// TIA Portal V17 export
// export: Created 2025-06-26T06:49:24.6875755Z, ExportSetting WithDefaults, DisplayName Totally Integrated Automation Portal, DisplayVersion V17 Update 8, DisplayName TIA Portal Openness, DisplayVersion V17 Update 8, DisplayName TIA Portal Version Control Interface, DisplayVersion V17, DisplayName STEP 7 Professional, DisplayVersion V17 Update 8, DisplayName STEP 7 Safety, DisplayVersion V17 Update 6, DisplayName WinCC Advanced, DisplayVersion V17 Update 8
DATA_BLOCK "DB_Alarms"   // DB44
{ S7_Optimized_Access := 'FALSE' }
AUTHOR : Heaten
VERSION : 0.1
// stored: AutoNumber true, DBAccessibleFromOPCUA true, DBAccessibleFromWebserver true, IsOnlyStoredInLoadMemory false, IsWriteProtectedInAS false
   VAR RETAIN
      bAckAll : Bool := FALSE;   // Global alarm acknowledge
      bCommonAlarm : Bool := FALSE;   // Global common alarm
      bCriticalAlarm : Bool := FALSE;   // Global critical alarm
      "0001_WatchdogTimeoutOB1" { S7_SetPoint := 'True'} : "stEvent";
      "0003_InitCurrentSettingsFailed" { S7_SetPoint := 'True'} : "stEvent";
      "1001_ConnectionToWinCClost" { S7_SetPoint := 'True'} : "stEvent";
      "1002_EmergencyStopActive" { S7_SetPoint := 'True'} : "stEvent";
      "1003_EmergencyStopResetFailed" { S7_SetPoint := 'True'} : "stEvent";
      "1004_HBL_PS_500_X2" { S7_SetPoint := 'True'} : "stEvent";
      "1101_HBL_SC_01_CommError" { S7_SetPoint := 'True'} : "stDigitalAlarm";
      "1102_HBL_SC_02_CommError" { S7_SetPoint := 'True'} : "stDigitalAlarm";
      "1103_HBL_SC_03_CommError" { S7_SetPoint := 'True'} : "stDigitalAlarm";
      "1110_HBL_SC_10_CommError" { S7_SetPoint := 'True'} : "stDigitalAlarm";
      "1121_HBL_SC_01_Tripped" { S7_SetPoint := 'True'} : "stDigitalAlarm";
      "1122_HBL_SC_02_Tripped" { S7_SetPoint := 'True'} : "stDigitalAlarm";
      "1123_HBL_SC_03_Tripped" { S7_SetPoint := 'True'} : "stDigitalAlarm";
      "1130_HBL_SC_10_Tripped" { S7_SetPoint := 'True'} : "stDigitalAlarm";
      "1140_HBL_SC_01_RunFailure" { S7_SetPoint := 'True'} : "stDigitalAlarm";
      "1142_HBL_SC_02_RunFailure" { S7_SetPoint := 'True'} : "stDigitalAlarm";
      "1143_HBL_SC_03_RunFailure" { S7_SetPoint := 'True'} : "stDigitalAlarm";
      "1150_HBL_SC_10_RunFailure" { S7_SetPoint := 'True'} : "stDigitalAlarm";
      "1201_HBL_PT_517_Fault" { S7_SetPoint := 'True'} : "stEvent";
      "1202_HBL_PT_612_Fault" { S7_SetPoint := 'True'} : "stEvent";
      "1203_HBL_PT_519_Fault" { S7_SetPoint := 'True'} : "stEvent";
      "1204_HBL_PT_544_Fault" { S7_SetPoint := 'True'} : "stEvent";
      "1205_HBL_TT_516_Fault" { S7_SetPoint := 'True'} : "stEvent";
      "1206_HBL_TT_611_Fault" { S7_SetPoint := 'True'} : "stEvent";
      "1207_HBL_TT_901_Fault" { S7_SetPoint := 'True'} : "stEvent";
      "1208_HBL_TT_518_Fault" { S7_SetPoint := 'True'} : "stEvent";
      "1209_HBL_HCV_576_A1_Fault" { S7_SetPoint := 'True'} : "stEvent";
      "1210_HBL_TT_573_Fault" { S7_SetPoint := 'True'} : "stEvent";
      "1212_HBL_TT_543_Fault" { S7_SetPoint := 'True'} : "stEvent";
      "1213_HBL_TT_546_Fault" { S7_SetPoint := 'True'} : "stEvent";
      "1214_HBL_TT_542_Fault" { S7_SetPoint := 'True'} : "stEvent";
      "1215_HBL_TT_571_Fault" { S7_SetPoint := 'True'} : "stEvent";
      "1216_HBL_TT_16_Fault" { S7_SetPoint := 'True'} : "stEvent";
      "1217_HBL_TT_17_Fault" { S7_SetPoint := 'True'} : "stEvent";
      "1218_HBL_TT_18_Fault" { S7_SetPoint := 'True'} : "stEvent";
      "1220_HBL_PT_960_Fault" { S7_SetPoint := 'True'} : "stEvent";
      "1221_HBL_PT_05_Fault" { S7_SetPoint := 'True'} : "stEvent";
      "1223_HBL_TT_03_Fault" { S7_SetPoint := 'True'} : "stEvent";
      "1224_HBL_TT_23_Fault" { S7_SetPoint := 'True'} : "stEvent";
      "1225_HBL_TT_24_Fault" { S7_SetPoint := 'True'} : "stEvent";
      "1226_HBL_TT_25_Fault" { S7_SetPoint := 'True'} : "stEvent";
      "1227_HBL_LT_610_Fault" { S7_SetPoint := 'True'} : "stEvent";
      "1228_HBL_TT_21_Fault" { S7_SetPoint := 'True'} : "stEvent";
      "1229_HBL_TT_22_Fault" { S7_SetPoint := 'True'} : "stEvent";
      "1230_HBL_LT_02_Fault" { S7_SetPoint := 'True'} : "stEvent";   // Deprecated
      "1231_HBL_HCV_578_A1_Fault" { S7_SetPoint := 'True'} : "stEvent";
      "1232_HBL_PT_503_Fault" { S7_SetPoint := 'True'} : "stEvent";
      "1233_HBL_TT_20_Fault" { S7_SetPoint := 'True'} : "stDigitalAlarm";
      "1234_HBL_PT_14_Fault" { S7_SetPoint := 'True'} : "stEvent";   // Deprecated
      "1235_HBL_PT_18_Fault" { S7_SetPoint := 'True'} : "stEvent";   // Deprecated
      "1236_HBL_PT_19_Fault" { S7_SetPoint := 'True'} : "stEvent";   // Deprecated
      "1237_HBL_PT_25_Fault" { S7_SetPoint := 'True'} : "stEvent";   // Deprecated
      "1238_HBL_TT_31_Fault" { S7_SetPoint := 'True'} : "stEvent";   // Deprecated
      "1239_HBL_TT_33_Fault" { S7_SetPoint := 'True'} : "stEvent";   // Deprecated
      "1240_HBL_TT_35_Fault" { S7_SetPoint := 'True'} : "stEvent";   // Deprecated
      "1241_HBL_HCV_576_Fault" { S7_SetPoint := 'True'} : "stEvent";
      "1242_HBL_HCV_578_Fault" { S7_SetPoint := 'True'} : "stEvent";
      "1243_HBL_PT_902_Fault" { S7_SetPoint := 'True'} : "stEvent";
      "1244_HBL_PT_572_Fault" { S7_SetPoint := 'True'} : "stEvent";
      "1245_HBL_PT_09_Fault" { S7_SetPoint := 'True'} : "stEvent";   // Deprecated
      "1246_HBL_PT_547_Fault" { S7_SetPoint := 'True'} : "stEvent";
      "1247_HBL_PT_541_Fault" { S7_SetPoint := 'True'} : "stEvent";
      "1248_HBL_PT_531_Fault" { S7_SetPoint := 'True'} : "stEvent";
      "1249_HBL_PT_701_Fault" { S7_SetPoint := 'True'} : "stEvent";
      "1251_HBL_PT_534_Fault" { S7_SetPoint := 'True'} : "stEvent";
      "1252_HBL_TT_540_Fault" { S7_SetPoint := 'True'} : "stEvent";
      "1253_HBL_TT_530_Fault" { S7_SetPoint := 'True'} : "stEvent";
      "1254_HBL_TT_533_Fault" { S7_SetPoint := 'True'} : "stEvent";
      "1255_HBL_CT_01_Fault" { S7_SetPoint := 'True'} : "stEvent";
      "1256_HBL_CT_615_Fault" { S7_SetPoint := 'True'} : "stEvent";
      "1257_HBL_CT_03_Fault" { S7_SetPoint := 'True'} : "stEvent";
      "1258_HBL_TT_26_Fault" { S7_SetPoint := 'True'} : "stEvent";
      "1259_HBL_TT_27_Fault" { S7_SetPoint := 'True'} : "stEvent";
      "1260_HBL_FT_520_Fault" { S7_SetPoint := 'True'} : "stEvent";
      "1262_HBL_TT_504_Fault" { S7_SetPoint := 'True'} : "stEvent";
      "1263_HBL_TT_34_Fault" { S7_SetPoint := 'True'} : "stEvent";
      "1264_HBL_PT_961_Fault" { S7_SetPoint := 'True'} : "stEvent";
      "1265_HBL_TT_502_Fault" { S7_SetPoint := 'True'} : "stEvent";
      "1266_HBL_LT_510_Fault" { S7_SetPoint := 'True'} : "stEvent";
      "1267_HBL_PT_511_Fault" { S7_SetPoint := 'True'} : "stEvent";
      "1268_HBL_TT_512_Fault" { S7_SetPoint := 'True'} : "stEvent";
      "1269_HBL_TT_532_Fault" { S7_SetPoint := 'True'} : "stEvent";
      "1270_HBL_AT_535_Fault" { S7_SetPoint := 'True'} : "stEvent";
      "1271_HBL_AT_545_Fault" { S7_SetPoint := 'True'} : "stEvent";
      "1272_HBL_PT_635_Fault" { S7_SetPoint := 'True'} : "stEvent";
      "1273_HBL_PT_636_Fault" { S7_SetPoint := 'True'} : "stEvent";
      "1274_HBL_LT_650_Fault" { S7_SetPoint := 'True'} : "stEvent";
      "1275_HBL_PT_651_Fault" { S7_SetPoint := 'True'} : "stEvent";
      "1276_HBL_PT_702_Fault" { S7_SetPoint := 'True'} : "stEvent";
      "1277_HBL_HCV_514_Fault" { S7_SetPoint := 'True'} : "stEvent";
      "1278_HBL_HCV_514_A1_Fault" { S7_SetPoint := 'True'} : "stEvent";
      "1279_HBL_HCV_515_Fault" { S7_SetPoint := 'True'} : "stEvent";
      "1280_HBL_HCV_515_A1_Fault" { S7_SetPoint := 'True'} : "stEvent";
      "1281_HBL_HCV_548_Fault" { S7_SetPoint := 'True'} : "stEvent";
      "1282_HBL_HCV_548_A1_Fault" { S7_SetPoint := 'True'} : "stEvent";
      "1283_HBL_HCV_575_Fault" { S7_SetPoint := 'True'} : "stEvent";
      "1284_HBL_HCV_575_A1_Fault" { S7_SetPoint := 'True'} : "stEvent";
      "1285_HBL_HCV_577_Fault" { S7_SetPoint := 'True'} : "stEvent";
      "1286_HBL_HCV_577_A1_Fault" { S7_SetPoint := 'True'} : "stEvent";
      "1287_HBL_HCV_579_Fault" { S7_SetPoint := 'True'} : "stEvent";
      "1288_HBL_HCV_579_A1_Fault" { S7_SetPoint := 'True'} : "stEvent";
      "1289_HBL_HCV_616_Fault" { S7_SetPoint := 'True'} : "stEvent";
      "1290_HBL_HCV_616_A1_Fault" { S7_SetPoint := 'True'} : "stEvent";
      "1291_HBL_HCV_700_Fault" { S7_SetPoint := 'True'} : "stEvent";
      "1292_HBL_HCV_700_A1_Fault" { S7_SetPoint := 'True'} : "stEvent";
      "1293_HBL_PT_618_Fault" { S7_SetPoint := 'True'} : "stEvent";
      "1294_HBL_LS_632_Fault" { S7_SetPoint := 'True'} : "stDigitalAlarm";
      "1295_HBL_LS_633_Fault" { S7_SetPoint := 'True'} : "stDigitalAlarm";
      "2018_HBL_PT_05_High" { S7_SetPoint := 'True'} : "stLimitAlarm";
      "2028_HBL_PT_17_Low" { S7_SetPoint := 'True'} : "stLimitAlarm";
      "2058_HBL_TT_03_Low" { S7_SetPoint := 'True'} : "stLimitAlarm";
      "2100_HBL_TT_03_High" { S7_SetPoint := 'True'} : "stLimitAlarm";
      "2101_HBL_TT_901_High" { S7_SetPoint := 'True'} : "stLimitAlarm";
      "2102_HBL_PT_503_High" { S7_SetPoint := 'True'} : "stLimitAlarm";
      "2103_HBL_TT_518_High" { S7_SetPoint := 'True'} : "stLimitAlarm";
      "2105_HBL_TT_546_High" { S7_SetPoint := 'True'} : "stLimitAlarm";
      "2106_HBL_TT_17_High" { S7_SetPoint := 'True'} : "stLimitAlarm";
      "2107_HBL_TT_16_High" { S7_SetPoint := 'True'} : "stLimitAlarm";
      "2108_HBL_TT_18_High" { S7_SetPoint := 'True'} : "stLimitAlarm";
      "2109_HBL_TT_20_High" { S7_SetPoint := 'True'} : "stLimitAlarm";
      "2110_HBL_TT_21_High" { S7_SetPoint := 'True'} : "stLimitAlarm";
      "2111_HBL_TT_22_High" { S7_SetPoint := 'True'} : "stLimitAlarm";
      "2112_HBL_LT_02_High" { S7_SetPoint := 'True'} : "stLimitAlarm";   // Deprecated
      "2113_HBL_CT_01_High" { S7_SetPoint := 'True'} : "stLimitAlarm";
      "2114_HBL_CT_615_High" { S7_SetPoint := 'True'} : "stLimitAlarm";
      "2115_HBL_PT_17_LowLow" { S7_SetPoint := 'True'} : "stLimitAlarm";
      "2116_HBL_PT_503_HighHigh" { S7_SetPoint := 'True'} : "stLimitAlarm";
      "2117_HBL_TT_542_Low" { S7_SetPoint := 'True'} : "stLimitAlarm";
      "2301_HeatSourceTempDropCritical" { S7_SetPoint := 'True'} : "stLimitAlarm";
      "2302_HeatSourceTempRiseCritical" { S7_SetPoint := 'True'} : "stLimitAlarm";
      "2303_SuperheatCompressor_High" { S7_SetPoint := 'True'} : "stLimitAlarm";
      "2304_SuperheatCompressor_Low" { S7_SetPoint := 'True'} : "stLimitAlarm";
      "2305_OilFilterDeltaP_High" { S7_SetPoint := 'True'} : "stLimitAlarm";
      "2306_OilFilterDeltaP_HighHigh" { S7_SetPoint := 'True'} : "stLimitAlarm";
      "2307_EvaporatorDischargePressureMeanValue" { S7_SetPoint := 'True'} : "stEvent";
      "2308_EvaporatorDischargePressureHigh" { S7_SetPoint := 'True'} : "stLimitAlarm";
      "2309_OilSeparatorStage1High" { S7_SetPoint := 'True'} : "stDigitalAlarm";
      "3020_SuperheatControlRegulatorFault" { S7_SetPoint := 'True'} : "stEvent";
      "3030_PinchControlRegulatorfault" { S7_SetPoint := 'True'} : "stEvent";
      "3400_HydrolockProtectionActive" { S7_SetPoint := 'True'} : "stEvent";
      "3401_DripPanLevelHigh" { S7_SetPoint := 'True'} : "stDigitalAlarm";
      "5000_OilHeatingActivationFailure" { S7_SetPoint := 'True'} : "stDigitalAlarm";
      "5001_OilHeatingDeactivationFailure" { S7_SetPoint := 'True'} : "stDigitalAlarm";
      "5200_CPC_LT_870_Fault" { S7_SetPoint := 'True'} : "stEvent";
      "5201_CPC_TT_871_Fault" { S7_SetPoint := 'True'} : "stEvent";
      "5202_CPC_PT_872_Fault" { S7_SetPoint := 'True'} : "stEvent";
      "5203_CPC_SC_01_CommError" { S7_SetPoint := 'True'} : "stDigitalAlarm";   // Deprecated
      "5204_CPC_SC_01_Tripped" { S7_SetPoint := 'True'} : "stDigitalAlarm";   // Deprecated
      "5205_CPC_LT_870_High" { S7_SetPoint := 'True'} : "stLimitAlarm";
      "5206_CPC_PT_862_Fault" { S7_SetPoint := 'True'} : "stEvent";
      "5250_SSC_TT_01_Fault" { S7_SetPoint := 'True'} : "stEvent";
      "5251_SSC_TT_02_Fault" { S7_SetPoint := 'True'} : "stEvent";
      "5252_SSC_TT_03_Fault" { S7_SetPoint := 'True'} : "stEvent";
      "5253_SSC_TT_04_Fault" { S7_SetPoint := 'True'} : "stEvent";
      "5254_SSC_PIT_01_Fault" { S7_SetPoint := 'True'} : "stEvent";
      "5255_SSC_PDT_01_Fault" { S7_SetPoint := 'True'} : "stEvent";
      "5256_SSC_LT_01_Fault" { S7_SetPoint := 'True'} : "stEvent";
      "5257_SSC_LT_01_Low" { S7_SetPoint := 'True'} : "stLimitAlarm";
      "5258_SSC_PDT_01_High" { S7_SetPoint := 'True'} : "stLimitAlarm";
      "5259_SSC_TT_02_High" { S7_SetPoint := 'True'} : "stLimitAlarm";
      "5260_SSC_TT_03_Low" { S7_SetPoint := 'True'} : "stLimitAlarm";
      "5261_SSC_PIT_01_Low" { S7_SetPoint := 'True'} : "stLimitAlarm";
      "5262_DeltaT_ShaftSealHigh" { S7_SetPoint := 'True'} : "stLimitAlarm";
      "5263_SSC_PIT_01_High" { S7_SetPoint := 'True'} : "stLimitAlarm";
      "5268_ShaftSealSystemShutdown" { S7_SetPoint := 'True'} : "stDigitalAlarm";
      "9023_HBL_HCV_576_Deviation" { S7_SetPoint := 'True'} : "stDeviationAlarm";
      "9024_HBL_HCV_578_Deviation" { S7_SetPoint := 'True'} : "stDeviationAlarm";
      "9025_HBL_HCV_577_Deviation" { S7_SetPoint := 'True'} : "stDeviationAlarm";
      "9026_HBL_HCV_579_Deviation" { S7_SetPoint := 'True'} : "stDeviationAlarm";
      "9027_HBL_HCV_575_Deviation" { S7_SetPoint := 'True'} : "stDeviationAlarm";
      "9028_HBL_HCV_616_Deviation" { S7_SetPoint := 'True'} : "stDeviationAlarm";
      "9029_HBL_HCV_700_Deviation" { S7_SetPoint := 'True'} : "stDeviationAlarm";
      "9030_HBL_HCV_514_Deviation" { S7_SetPoint := 'True'} : "stDeviationAlarm";
      "9031_HBL_HCV_548_Deviation" { S7_SetPoint := 'True'} : "stDeviationAlarm";
   END_VAR
BEGIN
   "0001_WatchdogTimeoutOB1".bEnable := true;
   "0003_InitCurrentSettingsFailed".bEnable := TRUE;
   "1001_ConnectionToWinCClost".bEnable := TRUE;
   "1002_EmergencyStopActive".bEnable := TRUE;
   "1003_EmergencyStopResetFailed".bEnable := TRUE;
   "1101_HBL_SC_01_CommError".bEnable := true;
   "1101_HBL_SC_01_CommError".bInput := FALSE;
   "1101_HBL_SC_01_CommError".tActivationDelay := T#1S;
   "1102_HBL_SC_02_CommError".bEnable := true;
   "1102_HBL_SC_02_CommError".tActivationDelay := T#1s;
   "1103_HBL_SC_03_CommError".bEnable := true;
   "1103_HBL_SC_03_CommError".tActivationDelay := T#1s;
   "1110_HBL_SC_10_CommError".bEnable := TRUE;
   "1110_HBL_SC_10_CommError".bInput := FALSE;
   "1110_HBL_SC_10_CommError".tActivationDelay := T#5s;
   "1121_HBL_SC_01_Tripped".bEnable := TRUE;
   "1121_HBL_SC_01_Tripped".bInput := FALSE;
   "1121_HBL_SC_01_Tripped".tActivationDelay := T#0MS;
   "1122_HBL_SC_02_Tripped".bEnable := true;
   "1122_HBL_SC_02_Tripped".tActivationDelay := T#0s;
   "1123_HBL_SC_03_Tripped".bEnable := true;
   "1130_HBL_SC_10_Tripped".bEnable := TRUE;
   "1130_HBL_SC_10_Tripped".bInput := FALSE;
   "1130_HBL_SC_10_Tripped".tActivationDelay := T#3s;
   "1140_HBL_SC_01_RunFailure".bEnable := TRUE;
   "1140_HBL_SC_01_RunFailure".bInput := FALSE;
   "1140_HBL_SC_01_RunFailure".tActivationDelay := T#0MS;
   "1142_HBL_SC_02_RunFailure".bEnable := true;
   "1142_HBL_SC_02_RunFailure".tActivationDelay := T#3s;
   "1143_HBL_SC_03_RunFailure".bEnable := true;
   "1143_HBL_SC_03_RunFailure".tActivationDelay := T#3s;
   "1150_HBL_SC_10_RunFailure".bEnable := TRUE;
   "1150_HBL_SC_10_RunFailure".bInput := FALSE;
   "1150_HBL_SC_10_RunFailure".tActivationDelay := T#3s;
   "1201_HBL_PT_517_Fault".bEnable := true;
   "1202_HBL_PT_612_Fault".bEnable := true;
   "1203_HBL_PT_519_Fault".bEnable := true;
   "1204_HBL_PT_544_Fault".bEnable := true;
   "1205_HBL_TT_516_Fault".bEnable := true;
   "1206_HBL_TT_611_Fault".bEnable := true;
   "1207_HBL_TT_901_Fault".bEnable := true;
   "1208_HBL_TT_518_Fault".bEnable := true;
   "1209_HBL_HCV_576_A1_Fault".bEnable := true;
   "1210_HBL_TT_573_Fault".bEnable := true;
   "1212_HBL_TT_543_Fault".bEnable := true;
   "1213_HBL_TT_546_Fault".bEnable := true;
   "1214_HBL_TT_542_Fault".bEnable := true;
   "1215_HBL_TT_571_Fault".bEnable := true;
   "1216_HBL_TT_16_Fault".bEnable := true;
   "1217_HBL_TT_17_Fault".bEnable := true;
   "1218_HBL_TT_18_Fault".bEnable := true;
   "1220_HBL_PT_960_Fault".bEnable := true;
   "1221_HBL_PT_05_Fault".bEnable := true;
   "1223_HBL_TT_03_Fault".bEnable := true;
   "1224_HBL_TT_23_Fault".bEnable := true;
   "1225_HBL_TT_24_Fault".bEnable := true;
   "1226_HBL_TT_25_Fault".bEnable := true;
   "1227_HBL_LT_610_Fault".bEnable := true;
   "1228_HBL_TT_21_Fault".bEnable := true;
   "1229_HBL_TT_22_Fault".bEnable := true;
   "1230_HBL_LT_02_Fault".bEnable := false;
   "1231_HBL_HCV_578_A1_Fault".bEnable := true;
   "1232_HBL_PT_503_Fault".bEnable := true;
   "1233_HBL_TT_20_Fault".bEnable := TRUE;
   "1233_HBL_TT_20_Fault".tActivationDelay := T#5S;
   "1234_HBL_PT_14_Fault".bEnable := true;
   "1235_HBL_PT_18_Fault".bEnable := true;
   "1236_HBL_PT_19_Fault".bEnable := true;
   "1237_HBL_PT_25_Fault".bEnable := false;
   "1238_HBL_TT_31_Fault".bEnable := true;
   "1239_HBL_TT_33_Fault".bEnable := true;
   "1240_HBL_TT_35_Fault".bEnable := true;
   "1241_HBL_HCV_576_Fault".bEnable := true;
   "1242_HBL_HCV_578_Fault".bEnable := true;
   "1243_HBL_PT_902_Fault".bEnable := true;
   "1244_HBL_PT_572_Fault".bEnable := true;
   "1245_HBL_PT_09_Fault".bEnable := true;
   "1246_HBL_PT_547_Fault".bEnable := true;
   "1247_HBL_PT_541_Fault".bEnable := true;
   "1248_HBL_PT_531_Fault".bEnable := true;
   "1249_HBL_PT_701_Fault".bEnable := true;
   "1251_HBL_PT_534_Fault".bEnable := true;
   "1252_HBL_TT_540_Fault".bEnable := true;
   "1253_HBL_TT_530_Fault".bEnable := true;
   "1254_HBL_TT_533_Fault".bEnable := true;
   "1255_HBL_CT_01_Fault".bEnable := true;
   "1256_HBL_CT_615_Fault".bEnable := true;
   "1258_HBL_TT_26_Fault".bEnable := true;
   "1259_HBL_TT_27_Fault".bEnable := true;
   "1260_HBL_FT_520_Fault".bEnable := true;
   "1262_HBL_TT_504_Fault".bEnable := true;
   "1263_HBL_TT_34_Fault".bEnable := true;
   "1264_HBL_PT_961_Fault".bEnable := true;
   "1265_HBL_TT_502_Fault".bEnable := true;
   "1266_HBL_LT_510_Fault".bEnable := true;
   "1267_HBL_PT_511_Fault".bEnable := true;
   "1268_HBL_TT_512_Fault".bEnable := true;
   "1269_HBL_TT_532_Fault".bEnable := true;
   "1270_HBL_AT_535_Fault".bEnable := true;
   "1271_HBL_AT_545_Fault".bEnable := true;
   "1272_HBL_PT_635_Fault".bEnable := true;
   "1273_HBL_PT_636_Fault".bEnable := true;
   "1274_HBL_LT_650_Fault".bEnable := true;
   "1275_HBL_PT_651_Fault".bEnable := true;
   "1276_HBL_PT_702_Fault".bEnable := true;
   "1283_HBL_HCV_575_Fault".bEnable := true;
   "1284_HBL_HCV_575_A1_Fault".bEnable := true;
   "1285_HBL_HCV_577_Fault".bEnable := true;
   "1286_HBL_HCV_577_A1_Fault".bEnable := true;
   "1287_HBL_HCV_579_Fault".bEnable := true;
   "1288_HBL_HCV_579_A1_Fault".bEnable := true;
   "1289_HBL_HCV_616_Fault".bEnable := true;
   "1290_HBL_HCV_616_A1_Fault".bEnable := true;
   "1291_HBL_HCV_700_Fault".bEnable := true;
   "1292_HBL_HCV_700_A1_Fault".bEnable := true;
   "1293_HBL_PT_618_Fault".bEnable := true;
   "1294_HBL_LS_632_Fault".tActivationDelay := t#5S;
   "2018_HBL_PT_05_High".bEnable := true;
   "2018_HBL_PT_05_High".fLimit := 1600.0;
   "2018_HBL_PT_05_High".fHysteresis := 0.0;
   "2018_HBL_PT_05_High".tActivationDelay := T#0MS;
   "2028_HBL_PT_17_Low".bEnable := true;
   "2028_HBL_PT_17_Low".fLimit := 30.0;
   "2028_HBL_PT_17_Low".fHysteresis := 0.0;
   "2028_HBL_PT_17_Low".tActivationDelay := T#30s;
   "2058_HBL_TT_03_Low".bEnable := true;
   "2058_HBL_TT_03_Low".fLimit := 0.0;
   "2058_HBL_TT_03_Low".fHysteresis := 1.0;
   "2058_HBL_TT_03_Low".tActivationDelay := T#180s;
   "2100_HBL_TT_03_High".bEnable := true;
   "2100_HBL_TT_03_High".tActivationDelay := T#0MS;
   "2101_HBL_TT_901_High".bEnable := true;
   "2101_HBL_TT_901_High".fHysteresis := 5.0;
   "2101_HBL_TT_901_High".tActivationDelay := T#5s;
   "2102_HBL_PT_503_High".bEnable := true;
   "2102_HBL_PT_503_High".tActivationDelay := T#1s;
   "2103_HBL_TT_518_High".bEnable := true;
   "2103_HBL_TT_518_High".tActivationDelay := T#1s;
   "2105_HBL_TT_546_High".bEnable := true;
   "2106_HBL_TT_17_High".bEnable := true;
   "2106_HBL_TT_17_High".tActivationDelay := T#10s;
   "2107_HBL_TT_16_High".bEnable := true;
   "2107_HBL_TT_16_High".tActivationDelay := T#10s;
   "2108_HBL_TT_18_High".bEnable := true;
   "2108_HBL_TT_18_High".tActivationDelay := T#10s;
   "2109_HBL_TT_20_High".bEnable := true;
   "2109_HBL_TT_20_High".tActivationDelay := T#0s;
   "2110_HBL_TT_21_High".bEnable := true;
   "2110_HBL_TT_21_High".fHysteresis := 5.0;
   "2110_HBL_TT_21_High".tActivationDelay := T#10s;
   "2111_HBL_TT_22_High".bEnable := true;
   "2111_HBL_TT_22_High".fHysteresis := 5.0;
   "2111_HBL_TT_22_High".tActivationDelay := T#10s;
   "2112_HBL_LT_02_High".bEnable := true;
   "2112_HBL_LT_02_High".tActivationDelay := T#5s;
   "2113_HBL_CT_01_High".bEnable := true;
   "2113_HBL_CT_01_High".fHysteresis := 50.0;
   "2114_HBL_CT_615_High".bEnable := true;
   "2114_HBL_CT_615_High".fHysteresis := 50.0;
   "2115_HBL_PT_17_LowLow".bEnable := true;
   // "2115_HBL_PT_17_LowLow".fLimit : Dynamic threshold!!
   "2115_HBL_PT_17_LowLow".tActivationDelay := T#2s;
   "2116_HBL_PT_503_HighHigh".bEnable := true;
   "2117_HBL_TT_542_Low".bEnable := true;
   "2117_HBL_TT_542_Low".fLimit := 5.0;
   "2117_HBL_TT_542_Low".fHysteresis := 1.0;
   "2117_HBL_TT_542_Low".tActivationDelay := T#2s;
   "2301_HeatSourceTempDropCritical".bEnable := true;
   "2302_HeatSourceTempRiseCritical".bEnable := true;
   "2303_SuperheatCompressor_High".bEnable := true;
   "2304_SuperheatCompressor_Low".bEnable := true;
   "2305_OilFilterDeltaP_High".bEnable := true;
   "2305_OilFilterDeltaP_High".fLimit := 30.0;
   "2305_OilFilterDeltaP_High".fHysteresis := 2.0;
   "2305_OilFilterDeltaP_High".tActivationDelay := T#10s;
   "2306_OilFilterDeltaP_HighHigh".bEnable := true;
   "2306_OilFilterDeltaP_HighHigh".fLimit := 100.0;
   "2306_OilFilterDeltaP_HighHigh".fHysteresis := 5.0;
   "2306_OilFilterDeltaP_HighHigh".tActivationDelay := T#5s;
   "2307_EvaporatorDischargePressureMeanValue".bEnable := true;
   "2308_EvaporatorDischargePressureHigh".bEnable := true;
   "2309_OilSeparatorStage1High".tActivationDelay := T#5m;
   "3020_SuperheatControlRegulatorFault".bEnable := true;
   "3400_HydrolockProtectionActive".bEnable := TRUE;
   "3401_DripPanLevelHigh".bEnable := false;
   "3401_DripPanLevelHigh".tActivationDelay := T#3S;
   "5000_OilHeatingActivationFailure".bEnable := TRUE;
   "5000_OilHeatingActivationFailure".bInput := FALSE;
   "5000_OilHeatingActivationFailure".tActivationDelay := T#2s;
   "5001_OilHeatingDeactivationFailure".bEnable := TRUE;
   "5001_OilHeatingDeactivationFailure".bInput := FALSE;
   "5001_OilHeatingDeactivationFailure".tActivationDelay := T#2s;
   "5200_CPC_LT_870_Fault".bEnable := true;
   "5201_CPC_TT_871_Fault".bEnable := true;
   "5202_CPC_PT_872_Fault".bEnable := true;
   "5203_CPC_SC_01_CommError".bEnable := false;
   "5203_CPC_SC_01_CommError".tActivationDelay := T#1S;
   "5204_CPC_SC_01_Tripped".bEnable := false;
   "5204_CPC_SC_01_Tripped".tActivationDelay := T#0MS;
   "5205_CPC_LT_870_High".bEnable := true;
   "5205_CPC_LT_870_High".fHysteresis := 2.0;
   "5205_CPC_LT_870_High".tActivationDelay := T#2S;
   "5206_CPC_PT_862_Fault".bEnable := true;
   "5250_SSC_TT_01_Fault".bEnable := true;
   "5251_SSC_TT_02_Fault".bEnable := true;
   "5252_SSC_TT_03_Fault".bEnable := true;
   "5253_SSC_TT_04_Fault".bEnable := true;
   "5254_SSC_PIT_01_Fault".bEnable := true;
   "5255_SSC_PDT_01_Fault".bEnable := true;
   "5256_SSC_LT_01_Fault".bEnable := true;
   "5257_SSC_LT_01_Low".bEnable := true;
   "5257_SSC_LT_01_Low".fLimit := 5.0;
   "5257_SSC_LT_01_Low".fHysteresis := 2.0;
   "5257_SSC_LT_01_Low".tActivationDelay := T#2S;
   "5258_SSC_PDT_01_High".bEnable := true;
   "5258_SSC_PDT_01_High".fLimit := 200.0;
   "5258_SSC_PDT_01_High".fHysteresis := 10.0;
   "5258_SSC_PDT_01_High".tActivationDelay := T#5S;
   "5259_SSC_TT_02_High".bEnable := true;
   "5259_SSC_TT_02_High".fLimit := 110.0;
   "5259_SSC_TT_02_High".fHysteresis := 2.0;
   "5259_SSC_TT_02_High".tActivationDelay := T#5S;
   "5260_SSC_TT_03_Low".bEnable := true;
   "5260_SSC_TT_03_Low".fLimit := 10.0;
   "5260_SSC_TT_03_Low".fHysteresis := 0.5;
   "5260_SSC_TT_03_Low".tActivationDelay := T#5S;
   "5261_SSC_PIT_01_Low".bEnable := true;
   "5261_SSC_PIT_01_Low".fLimit := 840.0;
   "5261_SSC_PIT_01_Low".fHysteresis := 10.0;
   "5261_SSC_PIT_01_Low".tActivationDelay := T#2S;
   "5262_DeltaT_ShaftSealHigh".bEnable := true;
   "5262_DeltaT_ShaftSealHigh".fLimit := 11.0;
   "5262_DeltaT_ShaftSealHigh".fHysteresis := 0.5;
   "5262_DeltaT_ShaftSealHigh".tActivationDelay := T#30S;
   "5263_SSC_PIT_01_High".bEnable := true;
   "5263_SSC_PIT_01_High".fLimit := 1400.0;
   "5263_SSC_PIT_01_High".fHysteresis := 5.0;
   "5263_SSC_PIT_01_High".tActivationDelay := T#2S;
   "5268_ShaftSealSystemShutdown".bEnable := false;
   "9023_HBL_HCV_576_Deviation".bEnable := true;
   "9023_HBL_HCV_576_Deviation".fDeviationLimit := 4.0;   // [%]
   "9023_HBL_HCV_576_Deviation".tActivationDelay := T#30s;
   "9024_HBL_HCV_578_Deviation".bEnable := true;
   "9024_HBL_HCV_578_Deviation".fDeviationLimit := 4.0;   // [%]
   "9024_HBL_HCV_578_Deviation".tActivationDelay := T#30s;
   "9025_HBL_HCV_577_Deviation".bEnable := true;
   "9025_HBL_HCV_577_Deviation".fDeviationLimit := 4.0;
   "9025_HBL_HCV_577_Deviation".tActivationDelay := T#30s;
   "9026_HBL_HCV_579_Deviation".bEnable := true;
   "9026_HBL_HCV_579_Deviation".fDeviationLimit := 4.0;
   "9026_HBL_HCV_579_Deviation".tActivationDelay := T#30s;
   "9027_HBL_HCV_575_Deviation".bEnable := true;
   "9027_HBL_HCV_575_Deviation".fDeviationLimit := 4.0;
   "9027_HBL_HCV_575_Deviation".tActivationDelay := T#5s;
   "9028_HBL_HCV_616_Deviation".bEnable := true;
   "9028_HBL_HCV_616_Deviation".fDeviationLimit := 4.0;
   "9028_HBL_HCV_616_Deviation".tActivationDelay := T#5s;
   "9029_HBL_HCV_700_Deviation".bEnable := true;
   "9029_HBL_HCV_700_Deviation".fDeviationLimit := 4.0;
   "9029_HBL_HCV_700_Deviation".tActivationDelay := T#5s;
   "9030_HBL_HCV_514_Deviation".bEnable := true;
   "9030_HBL_HCV_514_Deviation".fDeviationLimit := 4.0;
   "9030_HBL_HCV_514_Deviation".tActivationDelay := T#5s;
   "9031_HBL_HCV_548_Deviation".bEnable := true;
   "9031_HBL_HCV_548_Deviation".fDeviationLimit := 4.0;
   "9031_HBL_HCV_548_Deviation".tActivationDelay := T#5s;
END_DATA_BLOCK
